PROGRAM MAIN
VAR
	sMessage : STRING;
	iTestIndex : INT;
	GenAleatoire : Random;
	xTest : BOOL;
END_VAR;

// Premier test
CASE iTestIndex OF 
	1 : 
		sMessage := 'Bonjour jojo !';
	2 :
		sMessage := 'Au revoir';
	3 :
		sMessage :='';
END_CASE

// Second Test
IF iTestIndex = 0 THEN
	GenAleatoire(iMinVal := 1, iMaxVal := 10, o_iResult => iTestIndex);
ELSE
	// Do nothing
END_IF

END_PROGRAM

(* stored: Version 1.1.0.1, ProductVersion 3.1.4024.13
   POU MAIN: Id {f37ab39a-ee64-4305-b14b-001de0837e2a}, SpecialFunc None *)
